FUNCTION F_RAND : LREAL
VAR
	fbRand : DRAND;
END_VAR

fbRand(Seed := TO_INT(TIME()));
F_RAND := fbRand.Num;

END_FUNCTION

(* stored: Version 1.1.0.1, ProductVersion 3.1.4024.4
   POU F_RAND: Id {44073528-8af2-4251-a51f-0f280aef8209}, SpecialFunc None *)
